(* CoDeSys 2.3 export: ST_PumpProcessData.exp *)

(* Data type in Pump *)
(* ґРЭЭлХ ЯаЮжХббР ЭРбЮбР *)
TYPE ST_PumpProcessData :
STRUCT
    (* ёЧЬХапХЬлХ ЯРаРЬХвал *)
    rPressureInlet : REAL;      (* ґРТЫХЭШХ ЭР ТеЮФХ, СРа *)
    rPressureOutlet : REAL;     (* ґРТЫХЭШХ ЭР ТлеЮФХ, СРа *)
    rFlow : REAL;               (* АРбеЮФ, Ь?/з *)
    rTemperature : REAL;        (* ВХЬЯХаРвгаР, ?C *)
    
    (* їРаРЬХвал Юв їЗ *)
    rFrequency : REAL;          (* ЗРбвЮвР, іж *)
    rCurrent : REAL;            (* ВЮЪ, ° *)
    rPower : REAL;              (* јЮйЭЮбвм, ЪІв *)
    rSpeed : REAL;              (* БЪЮаЮбвм, ЮС/ЬШЭ *)
    
    (* АРбзХвЭлХ ЯРаРЬХвал *)
    rDifferentialPressure : REAL;  (* їХаХЯРФ ФРТЫХЭШп, СРа *)
    rHead : REAL;                   (* ЅРЯЮа, Ь *)
    rNPSHa : REAL;                  (* ґЮбвгЯЭлЩ ЪРТШвРжШЮЭЭлЩ ЧРЯРб, Ь *)
    rEfficiency : REAL;             (* єїґ, % *)
    rSpecificPower : REAL;          (* ГФХЫмЭРп ЬЮйЭЮбвм, ЪІв?з/Ь? *)
END_STRUCT
END_TYPE
